FUNCTION Convert_STRING_TO_TIME : Hresult
VAR_INPUT
	in : STRING;
	out : REFERENCE TO TIME;
END_VAR
VAR
	converted : TIME;
END_VAR

converted := STRING_TO_TIME(in);

IF (TIME_TO_STRING(converted) <> in) THEN
	Convert_STRING_TO_TIME := INCOMPATIBLE;
	RETURN;
END_IF

out := converted;

END_FUNCTION

(* stored: Version 1.1.0.1, ProductVersion 3.1.4024.12
   POU Convert_STRING_TO_TIME: Id {569e750b-938d-4456-8405-b7c78d692b33}, SpecialFunc None *)
